{attribute 'qualified_only'}
{attribute 'strict'}
TYPE JoystickState :
(
	NoCalib := 0,
	Operational := 1,
	Calib := 2
);
END_TYPE

(* stored: Version 1.1.0.1, ProductVersion 3.1.4022.18
   DUT JoystickState: Id {71825046-ba59-41b5-af7b-c2aa0e858b08} *)
